FUNCTION_BLOCK FB_ValveBACnet IMPLEMENTS I_Valve
VAR_INPUT
	//fbClient : FB_BACnet_Client;
END_VAR
VAR_OUTPUT
END_VAR
VAR
	//Properties
	bError 					: BOOL := FALSE;
	fOpeningActual 			: REAL;
	fOpeningSetpoint 		: REAL := 0;

(*	
	//BACnet parameters
	nPriority : BYTE := 12;
	
	//BACnet Mapping
	//Only one Client of the same DeviceInstance
*)
END_VAR

PROPERTY Error : BOOL
GET
Error := THIS^.bError;
END_GET
SET
THIS^.bError := Error;
END_SET
END_PROPERTY

PROPERTY OpeningActual : REAL
GET
OpeningActual := THIS^.fOpeningActual;
END_GET
SET
THIS^.fOpeningActual := OpeningActual;
END_SET
END_PROPERTY

PROPERTY OpeningSetpoint : REAL
GET
OpeningSetpoint := THIS^.fOpeningSetpoint;
END_GET
SET
THIS^.fOpeningSetpoint := OpeningSetpoint;
END_SET
END_PROPERTY

METHOD Run
(*
//Run BACnet client
fbClient();

//Read BACnet values
ReheaterValActBAC(fPresentValue=>fOpeningActual);

//Write BACnet values
ReheaterValSetBAC(fPV:=fOpeningSetpoint,bEnablePv:=TRUE,nPriority:=nPriority);
*)
END_METHOD

END_FUNCTION_BLOCK

(* stored: Version 1.1.0.1, ProductVersion 3.1.4024.0
   POU FB_ValveBACnet: Id {fbac7a6f-6bf1-4c62-bf13-aa77322e1ad6}, SpecialFunc None
   Property Error: Id {b622cc49-f082-48d2-a34b-232699e631f3}
   Get Get: Id {5e152892-1fe3-4d2d-ba3a-91400c750133}
   Set Set: Id {f664bff5-e8c4-42e2-9116-3346517e9ed1}
   Property OpeningActual: Id {bbd2e403-df54-4f37-9282-9e7c5daf91da}
   Get Get: Id {37041df0-9180-49a2-88ec-1f7ed50086c8}
   Set Set: Id {13cc65df-1f61-4914-af9d-043bac32b708}
   Property OpeningSetpoint: Id {2ff0074e-565b-4f4e-8913-c2d4f8f0d9f9}
   Get Get: Id {5ba05b76-37a9-4be7-ba2e-f0bfa7c8bb8a}
   Set Set: Id {9bdf2aca-2516-489d-a382-dfdcf83dcf27}
   Method Run: Id {f67494f0-daa5-4eab-a51c-88990ff06733} *)
